FUNCTION_BLOCK FB64
TITLE = 'process_F3'
AUTHOR : CB

VAR
	tmp : BOOL;
END_VAR


BEGIN


NETWORK
TITLE =
//
//	process/process_F3/SpinF1PROC
CALL FC63 (combE := 1);
CALL FB63,	DB63;
CALL FC63 (combE := 0);




END_FUNCTION_BLOCK
